FUNCTION_BLOCK E_SR_1 (* Event-driven bistable *)
  (* Standard: 61499-1 Annex A; Description: Copyright (c) 2017 fortiss GmbH This program and the accompanying materials are made available under the terms of the Eclipse Public License 2.0 which is available at https://www.eclipse.org/legal/epl-2.0/ SPDX-License-Identifier: EPL-2.0 *)
  (* Version 1.0, 2017-09-22, Alois Zoitl, fortiss GmbH, initial API and implementation and/or initial documentation *)
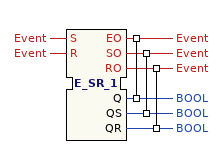
  EVENT_INPUT
    S; (* Set output Q *)
    R; (* Reset output Q *)
  END_EVENT
  EVENT_OUTPUT
    EO WITH Q; (* Output Q has changed *)
    SO WITH QS; (* Set output Q Operated *)
    RO WITH QR; (* Reset output Q operated *)
  END_EVENT
  VAR_OUTPUT
    Q : BOOL;
    QS : BOOL;
    QR : BOOL;
  END_VAR
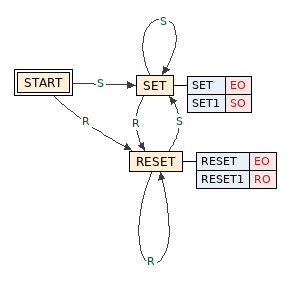
  EC_STATES
    START; (* Initial State *)
    SET : SET -> EO, SET1 -> SO;
    RESET : RESET -> EO, RESET1 -> RO;
  END_STATES
  EC_TRANSITIONS
    START TO SET := S;
    SET TO RESET := R;
    RESET TO SET := S;
    SET TO SET := S;
    RESET TO RESET := R;
    START TO RESET := R;
  END_TRANSITIONS
  ALGORITHM SET IN ST:
Q := TRUE;
  END_ALGORITHM
  ALGORITHM RESET IN ST:
Q := FALSE;
  END_ALGORITHM
  ALGORITHM SET1 IN ST:
QS := TRUE;
QR := FALSE;
  END_ALGORITHM
  ALGORITHM RESET1 IN ST:
QR := TRUE;
QS := FALSE;
  END_ALGORITHM
END_FUNCTION_BLOCK
